{attribute 'GeneratedUsingTerminal: EL1512-0000-0017'}
{attribute addProperty BoxType "EL1512-0000-0017"}
{attribute addProperty Id "Set_counter_doneBOOL1Counter_inhibitedBOOL1Status_of_input_clockBOOL1TxPDO_ToggleBOOL1"}
{attribute addProperty CRC "2328999243"}
{attribute addProperty Size "4"}
TYPE Status_8AD1B54B :
STRUCT
	{attribute addProperty Name "Set_counter_done"}
	Set_counter_done : BOOL;
	{attribute addProperty Name "Counter_inhibited"}
	Counter_inhibited : BOOL;
	{attribute addProperty Name "Status_of_input_clock"}
	Status_of_input_clock : BOOL;
	{attribute addProperty Name "TxPDO_Toggle"}
	TxPDO_Toggle : BOOL;
END_STRUCT
END_TYPE

(* stored: Version 1.2.0.0, ProductVersion 3.1.4024.9
   DUT Status_8AD1B54B: Id {643f0eaf-10cf-4f8a-9dde-bb60f77afb38} *)
